(* CoDeSys 2.3 export: VERSION.EXP *)

(* POU Version, ST *)
PROGRAM Version
VAR
(******************************************************************************************)
(* Version	Datum		Kommentar										*)
(* 1.00		29.08.2007	generated as a clone from UTIL_NO_REAL.LIB, removed POU CHARCURVE	 *)
(******************************************************************************************)
END_VAR
(* @TEXT_IMPLEMENTATION := 'ST' *)
;
END_PROGRAM
